// Mitsubishi GX Works2 project: n03   PLC: Q02/Q02H

PROGRAM MAIN
VAR
  자기_1 : 자기;
  자기_2 : 자기;
END_VAR
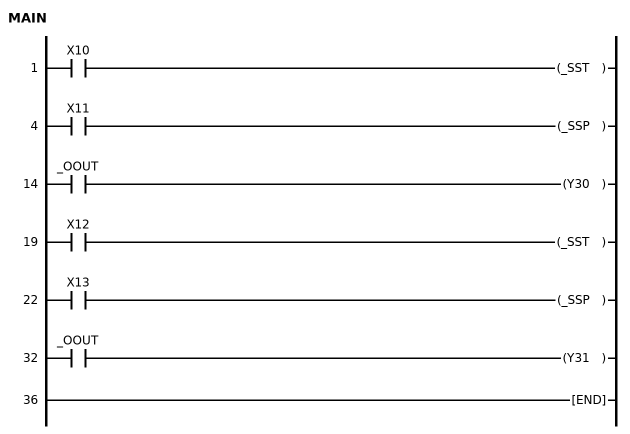
; FB BLK START 자기(자기_1)
1     LD      X10
      OUT     _SST
4     LD      X11
      OUT     _SSP
; FB START
; FB_NAME 자기
; INSTANCE_NAME 자기_1
; FB IN_B:SST
; FB OUT_OOUT:B
; FB IN_B:SSP
; FB END
14    LD      _OOUT
      OUT     Y30
; FB BLK END
; FB BLK START 자기(자기_2)
19    LD      X12
      OUT     _SST
22    LD      X13
      OUT     _SSP
; FB START
; FB_NAME 자기
; INSTANCE_NAME 자기_2
; FB IN_B:SST
; FB OUT_OOUT:B
; FB IN_B:SSP
; FB END
32    LD      _OOUT
      OUT     Y31
; FB BLK END
36    END
END_PROGRAM

FUNCTION_BLOCK 자기
VAR_INPUT
  SST : BOOL;
  SSP : BOOL;
END_VAR
VAR_OUTPUT
  OOUT : BOOL;
END_VAR
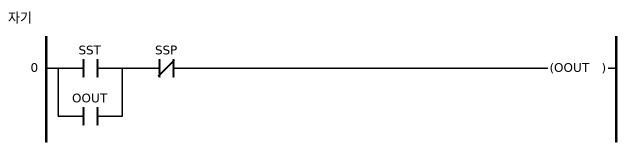
0     LD      SST
      OR      OOUT
      ANI     SSP
      OUT     OOUT
END_FUNCTION_BLOCK
